ACTION POSTRUN:
(******************************************************************************)
(********** Release of PostRun - Move System to Shutdown task   ***************)
(******************************************************************************)
CallPostRunNr_no_u16 := CallPostRunNr_no_u16 + 1;

(* Release Postrun after 5 sec *)
IF (CallPostRunNr_no_u16 > 500) THEN
    bds_sys_releasePostRunProlong(); (* transitions system state from POSTRUN to SHUTDOWN *)
END_IF
END_ACTION

ACTION READ_PARAMETERS:
(******************************************************************************)
(************************ Debug Manager  **************************************)
(******************************************************************************)
PRG_DebugManager();
(******************************************************************************)
(************************ NVM Config.  ****************************************)
(******************************************************************************)
PRG_NVMConfig();
END_ACTION

ACTION RUN:
(******************************************************************************)
(**************************** CAN Wakeup Handling   ***************************)
(******************************************************************************)
(* resetInfo_s.rbr_UserDefined_u32 = 0x01 means that the Wakeup has happened via CAN via CAN Channel 1 *)
(* resetInfo_s.rbr_UserDefined_u32 = 0x04 means that the Wakeup has happened via CAN via CAN Channel 4 *)
IF ((16#01 = INIT_PRG.ResetInfo_struc.rbr_UserDefined_u32) OR (16#04 = INIT_PRG.ResetInfo_struc.rbr_UserDefined_u32)) THEN
    bds_sys_cancelAltWakeup(); (* forces system state to go to POSTRUN *)
END_IF
END_ACTION

ACTION STARTLOCK:
StartRelease_st_b := TRUE;
END_ACTION

END_PROGRAM

// BODAS_RC18_12_40/Application/01 MainTask/03 Communication/00 CAN/PRG_CANOut
(*********************************************************************************************************************
 *     __   __   ___  ___           __   __        __   __  ___
 *   /_ / /  / /__  /    /__/     /_ / /_   |_ / /_ / /  /  /  /__/
 *  /__/ /__/ __ / /__  /  /     /  | /__  /  | /  | /__/  /  /  /
 *
 * Project: Hello World for ml290.rts
 *
 * Program: PRG_CANOut
 *
 * Author:  
 *
 * Description:
 * Interface for CAN Transmitting
 *
 * (c) Copyright by BOSCH REXROTH AG, all rights reserved
 *
 *********************************************************************************************************************)
PROGRAM PRG_CANOut
VAR
    (* Buffer for rx databoxes *)
    CAN1RxData_astruc   : ARRAY[1..2] OF bds_can_DataboxData_ts;
    CAN2RxData_astruc   : ARRAY[1..5] OF bds_can_DataboxData_ts;
    bds_IPduGrpVctr_au8 : ARRAY[0..7] OF USINT;
    retSet_u16          : UINT;
    retStrt_u16         : UINT;
    data_au8            : ARRAY[1..8] OF USINT;
    dataTx_au8          : ARRAY[1..8] OF USINT; (* data ARRAY FOR CAN legacy data*)
    sigData_au8         : ARRAY[1..8] OF USINT; (* data ARRAY FOR CAN signal based data*)
END_VAR
VAR_INPUT
    i_statusNvmIni_u16  : UINT;
    i_iPmpFwdAct_mA_u16 : UINT;
    i_iPmpFwdSet_mA_u16 : UINT;
    i_CtrlValve_u8      : USINT;
    i_rxActEngPercTq_u8 : USINT;
    i_vWhlSpd_kph_u16   : INT;
    i_uPmpSnsr_mV_u16   : UINT;
    i_frqVehSnsr_Hz_u32 : UDINT;
    i_anValue_perc_u8   : USINT;
    i_stBrkSwt_u8       : USINT;
END_VAR
VAR_OUTPUT
END_VAR

(* ----------------------------------------------------------------------- *)
(* --- CAN legacy transmit --- *)
(* ----------------------------------------------------------------------- *)
(* Send a cyclic STD CAN message ON CAN1 when in OsMain *)
bds_can_sendData(bds_can_Chnl_te.BDS_CAN_1_D, 16#2, BDS_CAN_STD_DU8, 0, 0);
(* SnsrInp1 Tx *)
dataTx_au8[1] := UINT_TO_USINT(i_uPmpSnsr_mV_u16);
dataTx_au8[2] := UINT_TO_USINT(SHR(i_uPmpSnsr_mV_u16, 8));
dataTx_au8[3] := i_stBrkSwt_u8;
dataTx_au8[4] := UDINT_TO_USINT(i_frqVehSnsr_Hz_u32);
dataTx_au8[5] := UDINT_TO_USINT(SHR(i_frqVehSnsr_Hz_u32, 8));
dataTx_au8[6] := UDINT_TO_USINT(SHR(i_frqVehSnsr_Hz_u32, 16));
dataTx_au8[7] := UDINT_TO_USINT(SHR(i_frqVehSnsr_Hz_u32, 24));
dataTx_au8[8] := i_anValue_perc_u8; (* to test if 0x18FF1128 is received - legacy*)

IF (0 = bds_can_sendData(bds_can_Chnl_te.BDS_CAN_2_D, 16#18FF2703, BDS_CAN_EXD_DU8, 8, ADR(dataTx_au8))) THEN
    (* ok, message is buffered and will be sent as fast as possible *)
    ;
END_IF

(* ELSE: error *)
(* Outp1 Tx message from CAN dbc *)
(* Output currents *)
dataTx_au8[1] := UINT_TO_USINT(i_iPmpFwdAct_mA_u16);         (* LSB *)
dataTx_au8[2] := UINT_TO_USINT(SHR(i_iPmpFwdAct_mA_u16, 8)); (* MSB *)
dataTx_au8[3] := UINT_TO_USINT(i_iPmpFwdSet_mA_u16);
dataTx_au8[4] := UINT_TO_USINT(SHR(i_iPmpFwdSet_mA_u16, 8));
dataTx_au8[5] := i_CtrlValve_u8;
dataTx_au8[6] := TO_USINT(GlobalVariables.PrmAsw_gstruc.listCtrlVlv_enu);                   (* to test if the list DID C002 is received *)
dataTx_au8[7] := TO_USINT(INT_TO_WORD(GlobalVariables.PrmAsw_gstruc.nrCogs_s16) AND 16#FF); (* to test if the no. of cogs DID C003 is received *)
dataTx_au8[8] :=
    i_rxActEngPercTq_u8; (* to test if ComConf_ComSignal_ComSignal_ActualEngPercentTorque_xRx is received *)

IF (0 = bds_can_sendData(bds_can_Chnl_te.BDS_CAN_2_D, 16#18FF2603, BDS_CAN_EXD_DU8, 8, ADR(dataTx_au8))) THEN
    (* ok, message is buffered and will be sent as fast as possible *)
    ;
END_IF

(* else: error *)
(* ----------------------------------------------------------------------- *)
(* --- CAN signal based transmit --- *)
(* ----------------------------------------------------------------------- *)
(* CCVS message FROM CAN dbc - out OF the 100 ms loop *)
(* Vehicle Speed *)
sigData_au8[1] := UINT_TO_USINT(i_vWhlSpd_kph_u16);
sigData_au8[2] := UINT_TO_USINT(SHR(i_vWhlSpd_kph_u16, 8));

IF (0 = bds_can_sendSignal(ComConf_ComSignal_ComSignal_WheelBasedVehicleSpeed_xTx, ADR(sigData_au8), 0)) THEN
    (* ok,message is sent on bus with updated signal data *)
    ;
END_IF

(* Parking Brake (Control Valve) *)
sigData_au8[1] := i_CtrlValve_u8;

IF (0 = bds_can_sendSignal(ComConf_ComSignal_ComSignal_ParkingBrakeSwitch_xTx, ADR(sigData_au8), 0)) THEN
    (* ok,message is sent on bus with updated signal data *)
    ;
END_IF

END_PROGRAM

// BODAS_RC18_12_40/Application/01 MainTask/11 Parameters/Programs/PRG_NVMConfig
(*********************************************************************************************************************
 *     __   __   ___  ___           __   __        __   __  ___
 *   /_ / /  / /__  /    /__/     /_ / /_   |_ / /_ / /  /  /  /__/
 *  /__/ /__/ __ / /__  /  /     /  | /__  /  | /  | /__/  /  /  /
 *
 * Project: Hello World for ml290.rts
 *
 * Program: PRG_NVMConfig
 *
 * Author:  
 *
 * Description:
 * Interface for Paramters
 *
 * (c) Copyright by BOSCH REXROTH AG, all rights reserved
 *
 *********************************************************************************************************************)
PROGRAM PRG_NVMConfig
VAR
    status_u16 : UINT;
END_VAR

;

END_PROGRAM

// BODAS_RC18_12_40/Application/01 MainTask/02 Outputs/PRG_Outputs
(*********************************************************************************************************************
*    __   __   ___  ___           __   __        __   __  ___
*   /_ / /  / /__  /    /__/     /_ / /_   |_ / /_ / /  /  /  /__/
*  /__/ /__/ __ / /__  /  /     /  | /__  /  | /  | /__/  /  /  /
*
* Project: Hello World for ml290.rts
*
* Program: PRG_Outputs
*
* Author: 
*
* Description:
* Interface for the hardware outputs to the application
*
* (c) Copyright by BOSCH REXROTH AG, all rights reserved
*
*********************************************************************************************************************)
PROGRAM PRG_Outputs
VAR_INPUT
    i_UPumpSensr_mV_u16 : UINT;
END_VAR
VAR
    diagParam_s             : bds_outCmn_diagParam_ts;
    bds_outPwm_retGet_s     : bds_outPwm_get_ts; (* PWM output status *)
    no_UBatt_mV_u16         : UINT;
    st_FlgInhActive_b       : BOOL;
    st_FlgUBatLowDetd_b     : BOOL;
    st_FlgUBatLowDetdPrev_b : BOOL;
    st_FlgOutpLocked_b      : BOOL;
    st_FlgUnderUbat_b       : BOOL;
    st_FlgRstInh_b          : BOOL;
    st_FlgRstLowBatt_b      : BOOL;
    no_NrCycDebRst_u16      : UINT;
    no_CurrentK07_mA_u16    : UINT;
    iPmpFwdSet_mA_u16       : UINT;
    st_CurStK07_u8          : USINT;
    no_UPumpSensr_mV_u16    : UINT;
    st_CtrlValve_u8         : USINT;
    st_BrkSwt_u8            : USINT;
    MngInh_struc            : struc_MngInhb;
    PHMDL_CHNL1             : UINT := (UDINT_TO_UINT(PHMDL) OR UDINT_TO_UINT(CHNL1));
END_VAR
VAR CONSTANT
    st_ENotOk_cby    : BYTE := 16#01;
    st_StdHigh_cby   : BYTE := 16#01;
    st_StdLow_cby    : BYTE := 16#00;
    st_StdActive_cby : BYTE := 16#01;
    st_StdIdle_cby   : BYTE := 16#00;
    st_StdOn_cby     : BYTE := 16#00;
    st_StdOff_cby    : BYTE := 16#01;
END_VAR

(* Inhibit handling *)
ACT_HandleInhibit();
(* PropValve - read actual current *)
bds_outPwm_retGet_s := bds_outPwm_get(bds_outPwm_signal_te.bds_outPwm_K07_E);

(* check return state of BDS-Function call *)
IF (bds_outCmn_ok_E = bds_outPwm_retGet_s.statusApi_e) THEN
    (* Call successful, signal is valid *)
    ;
ELSE
    (* error handling *)
    no_CurrentK07_mA_u16 := bds_outPwm_retGet_s.iAct_mA_u16;
END_IF

(* Calculate set current *)
(* PropValve [K07]= PmpSensor [K52] * Factor [parameter DID 0xC001] *)
iPmpFwdSet_mA_u16 := i_UPumpSensr_mV_u16 * INT_TO_UINT(GlobalVariables.PrmAsw_gstruc.fctPmp_s16);

(* Calculate set state *)
(* CtrlValve [K12] = BrkSwitch [K78] | List [DID 0xC002] *)
CASE (GlobalVariables.PrmAsw_gstruc.listCtrlVlv_enu) OF
enu_listCtrlVlv.st_fctOff_cenu: st_CtrlValve_u8   := st_StdIdle_cby;
enu_listCtrlVlv.st_fctOnPos_cenu: st_CtrlValve_u8 := st_BrkSwt_u8;
enu_listCtrlVlv.st_fctOnNeg_cenu: IF (NOT (0 = st_BrkSwt_u8)) THEN
        st_CtrlValve_u8 := st_StdIdle_cby;
    ELSE
        st_CtrlValve_u8 := st_StdActive_cby;
    END_IF
    ELSE
        ;
END_CASE

(* ----------------------------------------------------------------------- *)
(* --- Set outputs ---*)
(* ----------------------------------------------------------------------- *)
(* Set outputs only when inhibit is not active *)
(* PropValve *)
bds_outPwm_cfgMode(bds_outPwm_signal_te.bds_outPwm_K07_E, bds_outMode_CLCC_E);   (* Configure K07 as closed loop current control *)
bds_outPwm_setCurrent(bds_outPwm_signal_te.bds_outPwm_K07_E, iPmpFwdSet_mA_u16); (* Set current set point for proportional valve *)
(* CtrlValve *)
bds_outDig_set(bds_outDig_signal_te.bds_outDig_K13_E, (st_CtrlValve_u8 > 0));
(* Safout *)
bds_out_po_cfg(bds_out_po_signal_te.K09, STD_ON);                                                (* Configure K09 as closed loop current control *)
bds_out_po_cfg(bds_out_po_signal_te.K73, STD_ON);                                                (* Configure K73 as closed loop current control *)
bds_safout(PHMDL_CHNL1, bds_out_po_signal_te.K09, GlobalVariables.PrmAsw_gstruc.iSpSafout1_u16); (* Safout - HS1 *)
bds_safout(PHMDL_CHNL1, bds_out_po_signal_te.K73, GlobalVariables.PrmAsw_gstruc.iSpSafout2_u16); (* Safout - HS2 *)

ACTION ACT_HandleInhibit:
(* Monitor battery voltage AND state OF inhibit            *
 * reset inhibit in CASE it was activated BY under voltage *
*)
(* Invert logic of flgStInhb_u8 *)
st_FlgInhActive_b := NOT( PRG_Inputs.st_FlgStInhb_u8 > 0 );

bds_sys_aiv(bds_sys_aiv_signal_te.UBAT_MON, ADR(no_UBatt_mV_u16));  (* battery supply voltage *)   

IF( no_UBatt_mV_u16 < 7000 ) THEN (* under voltage detection if the battery voltage is less than 7V *)
  st_FlgUnderUbat_b := TRUE;
END_IF
      
st_FlgUBatLowDetd_b := ( ( st_FlgInhActive_b )OR (6500  >  no_UBatt_mV_u16 ) );

(* Inhibit Reset (i.e. release outputs again after emergency stop) *)
st_FlgRstInh_b :=	st_FlgInhActive_b                   AND  (* Inhibit is active -> Outputs are disabled *)
					( 9000 <  no_UBatt_mV_u16 )         AND  (* Voltage is greater than x V *)
					( 0    =  PRG_Inputs.st_K21Inh_u8 ) AND  (* Inhibit inputs are in a legitimate state *)
					( 0    <> PRG_Inputs.st_K22Inh_u8 );     (* Inhibit inputs are in a legitimate state *)
					
(* Low Battery Reset (i.e. release outputs after low battery was detected) *)
st_FlgRstLowBatt_b :=	st_FlgInhActive_b           AND  (* Inhibit is not active *)  
						st_FlgOutpLocked_b          AND  (* Outputs are locked *)
						( 9000 < no_UBatt_mV_u16 );      (* Voltage is greater than x V *)
						
						
(* Debounce Reset *)
IF( st_FlgRstInh_b OR st_FlgRstLowBatt_b ) THEN  
	no_NrCycDebRst_u16 := no_NrCycDebRst_u16 + 1;
END_IF					


IF( 5 < no_NrCycDebRst_u16 ) THEN
	(* Reset inhibit (enables the output again) *)	
	bds_sys_resetINH();
	
	(* Re-Configure K08 as power supply FOR K13 Control valve *)
	diagParam_s.diFullDiag_l     := TRUE;
	diagParam_s.diCntlAndDiag_l  := FALSE;
	diagParam_s.diOpenLoadDetn_l := TRUE;
	diagParam_s.diNonHotSCDetn_l := FALSE;
	
	bds_outPwm_cfgDiag(bds_outPwm_signal_te.bds_outPwm_K08_E, diagParam_s);
	bds_outPwm_setDutyCycle(bds_outPwm_signal_te.bds_outPwm_K08_E, 1000);
	
	st_FlgUnderUbat_b  := FALSE;
	no_NrCycDebRst_u16 := 0;

ELSE
	;	
END_IF
END_ACTION

ACTION ACT_InitOutputs:
diagParam_s.diCntlAndDiag_l := TRUE; (* disable outputs *)
(* Disable unused proportional outputs *)
(*bds_outPwm_cfgDiag(bds_outPwm_signal_te.bds_outPwm_K07_E, diagParam_s);*) (* used FOR PropValve *)
(*bds_outPwm_cfgDiag(bds_outPwm_signal_te.bds_outPwm_K09_E, diagParam_s);*) (* Safout HS1 *)
(*bds_outPwm_cfgDiag(bds_outPwm_signal_te.bds_outPwm_K73_E, diagParam_s);*) (* Safout HS2 *)
(*bds_outPwm_cfgDiag(bds_outPwm_signal_te.bds_outPwm_K08_E, diagParam_s);*) (* used as power supply for Control valve *)
bds_outPwm_cfgDiag(bds_outPwm_signal_te.bds_outPwm_K29_E, diagParam_s);
bds_outPwm_cfgDiag(bds_outPwm_signal_te.bds_outPwm_K17_E, diagParam_s);
bds_outPwm_cfgDiag(bds_outPwm_signal_te.bds_outPwm_A32_E, diagParam_s);
bds_outPwm_cfgDiag(bds_outPwm_signal_te.bds_outPwm_A47_E, diagParam_s);
bds_outPwm_cfgDiag(bds_outPwm_signal_te.bds_outPwm_A31_E, diagParam_s);
bds_outPwm_cfgDiag(bds_outPwm_signal_te.bds_outPwm_A48_E, diagParam_s);
bds_outPwm_cfgDiag(bds_outPwm_signal_te.bds_outPwm_A46_E, diagParam_s);
bds_outPwm_cfgDiag(bds_outPwm_signal_te.bds_outPwm_A33_E, diagParam_s);
bds_outPwm_cfgDiag(bds_outPwm_signal_te.bds_outPwm_A34_E, diagParam_s);
bds_outPwm_cfgDiag(bds_outPwm_signal_te.bds_outPwm_A51_E, diagParam_s);
bds_outPwm_cfgDiag(bds_outPwm_signal_te.bds_outPwm_A35_E, diagParam_s);
bds_outPwm_cfgDiag(bds_outPwm_signal_te.bds_outPwm_A53_E, diagParam_s);
bds_outPwm_cfgDiag(bds_outPwm_signal_te.bds_outPwm_A52_E, diagParam_s);
bds_outPwm_cfgDiag(bds_outPwm_signal_te.bds_outPwm_A54_E, diagParam_s);
bds_outPwm_cfgDiag(bds_outPwm_signal_te.bds_outPwm_K16_E, diagParam_s);
(*bds_outPwm_cfgDiag(bds_outPwm_signal_te.bds_outPwm_K14_E, diagParam_s);*) (* Safout LS *)
bds_outPwm_cfgDiag(bds_outPwm_signal_te.bds_outPwm_K15_E, diagParam_s);
bds_outPwm_cfgDiag(bds_outPwm_signal_te.bds_outPwm_A19_E, diagParam_s);
bds_outPwm_cfgDiag(bds_outPwm_signal_te.bds_outPwm_A05_E, diagParam_s);
bds_outPwm_cfgDiag(bds_outPwm_signal_te.bds_outPwm_A20_E, diagParam_s);
bds_outPwm_cfgDiag(bds_outPwm_signal_te.bds_outPwm_A09_E, diagParam_s);
bds_outPwm_cfgDiag(bds_outPwm_signal_te.bds_outPwm_A02_E, diagParam_s);
bds_outPwm_cfgDiag(bds_outPwm_signal_te.bds_outPwm_A17_E, diagParam_s);
bds_outPwm_cfgDiag(bds_outPwm_signal_te.bds_outPwm_K51_E, diagParam_s);
bds_outPwm_cfgDiag(bds_outPwm_signal_te.bds_outPwm_K12_E, diagParam_s);
bds_outPwm_cfgDiag(bds_outPwm_signal_te.bds_outPwm_A03_E, diagParam_s);
bds_outPwm_cfgDiag(bds_outPwm_signal_te.bds_outPwm_A18_E, diagParam_s);
bds_outPwm_cfgDiag(bds_outPwm_signal_te.bds_outPwm_A08_E, diagParam_s);
bds_outPwm_cfgDiag(bds_outPwm_signal_te.bds_outPwm_A07_E, diagParam_s);
bds_outPwm_cfgDiag(bds_outPwm_signal_te.bds_outPwm_K80_E, diagParam_s);
bds_outPwm_cfgDiag(bds_outPwm_signal_te.bds_outPwm_K81_E, diagParam_s);
bds_outPwm_cfgDiag(bds_outPwm_signal_te.bds_outPwm_K82_E, diagParam_s);
bds_outPwm_cfgDiag(bds_outPwm_signal_te.bds_outPwm_K83_E, diagParam_s);
(* Disable unused digital outputs *)
(*bds_outDig_cfgDiag(bds_outDig_K13_E, diagParam_s);*) (* used for CtrlValve *)
bds_outDig_cfgDiag(bds_outDig_signal_te.bds_outDig_A04_E, diagParam_s);
bds_outDig_cfgDiag(bds_outDig_signal_te.bds_outDig_A10_E, diagParam_s);
bds_outDig_cfgDiag(bds_outDig_signal_te.bds_outDig_A50_E, diagParam_s);
bds_outDig_cfgDiag(bds_outDig_signal_te.bds_outDig_A56_E, diagParam_s);
bds_outDig_cfgDiag(bds_outDig_signal_te.bds_outDig_A11_E, diagParam_s);
bds_outDig_cfgDiag(bds_outDig_signal_te.bds_outDig_A55_E, diagParam_s);
bds_outDig_cfgDiag(bds_outDig_signal_te.bds_outDig_A01_E, diagParam_s);
bds_outDig_cfgDiag(bds_outDig_signal_te.bds_outDig_A06_E, diagParam_s);
bds_outDig_cfgDiag(bds_outDig_signal_te.bds_outDig_A16_E, diagParam_s);
bds_outDig_cfgDiag(bds_outDig_signal_te.bds_outDig_A58_E, diagParam_s);
bds_outDig_cfgDiag(bds_outDig_signal_te.bds_outDig_A49_E, diagParam_s);
bds_outDig_cfgDiag(bds_outDig_signal_te.bds_outDig_K84_E, diagParam_s);
bds_outDig_cfgDiag(bds_outDig_signal_te.bds_outDig_K85_E, diagParam_s);
bds_outDig_cfgDiag(bds_outDig_signal_te.bds_outDig_K86_E, diagParam_s);
bds_outDig_cfgDiag(bds_outDig_signal_te.bds_outDig_K87_E, diagParam_s); (* for the visualisation in BODAS-service App --> I/O *)
(* Configure K08 as power supply for K13 Control valve *)
diagParam_s.diFullDiag_l     := TRUE;
diagParam_s.diCntlAndDiag_l  := FALSE;
diagParam_s.diOpenLoadDetn_l := TRUE;
diagParam_s.diNonHotSCDetn_l := FALSE;
bds_outPwm_cfgDiag(bds_outPwm_signal_te.bds_outPwm_K08_E, diagParam_s);
bds_outPwm_setDutyCycle(bds_outPwm_signal_te.bds_outPwm_K08_E, 1000);
END_ACTION

END_PROGRAM

// BODAS_RC18_12_40/Application/01 MainTask/01 Inputs/PRG_Inputs
(*********************************************************************************************************************
 *     __   __   ___  ___           __   __        __   __  ___
 *   /_ / /  / /__  /    /__/     /_ / /_   |_ / /_ / /  /  /  /__/
 *  /__/ /__/ __ / /__  /  /     /  | /__  /  | /  | /__/  /  /  /
 *
 * Project: Hello World for ml290.rts
 *
 * Program: PRG_Inputs
 *
 * Author:  
 *
 * Description:
 * Interface for the hardware inputs to the application
 *
 * (c) Copyright by BOSCH REXROTH AG, all rights reserved
 *
 *********************************************************************************************************************)
PROGRAM PRG_Inputs
VAR_INPUT
    i_TaskCycleTime_ms_u16 : UINT;
END_VAR
VAR
    st_K21Inh_u8           : USINT;
    st_K22Inh_u8           : USINT;
    st_FlgStInhb_u8        : USINT;
    bds_inPwm_getFrqPwm_s  : bds_inPwm_frqMeasmt_ts;
    FrqP_Hz_10_u32         : UDINT;                (* frequency [0.1Hz] *)
    Tmp_u32                : UDINT;                (* temporary *)
    stPmpSnsrU_struc       : bds_inU_measmt_ts;    (*structure FOR Pump sensor voltage measurement *)
    uPmpSnsr_mV_u16        : UINT;                 (* voltage [mV], ECU pin K52 *)
    stPmpSnsrSigInvldErr_e : bds_dsmCmn_fltLvl_te; (* status of error: PmpSnsr *)
    (* K78 � DIG, BrkSwitch - read as AIV *)
    stBrkSwtU_struc       : bds_inU_measmt_ts;    (* structure FOR Brake switch voltage measurement *)
    uBrkSwt_mV_u16        : UINT;                 (* voltage [mV], ECU pin K78 *)
    stBrkSwt_u8           : USINT;                (* status OF break switch, ECU pin K78 *)
    stBrkSwtSigInvldErr_e : bds_dsmCmn_fltLvl_te; (* status OF error: BrkSwt *)
    (* K54_VI � FREQ, VehSensor *)
    stVehSnsrFrq_struc : bds_inPwm_frqMeasmt_ts; (*structure FOR vehicle sensor frequency measurement *)
    frqVehSnsr_Hz_u32  : UDINT;                  (* frequency [Hz], ECU pin K54_VI *)
    vWhlSpd_kph_u16    : UINT;                   (* vehicle speed [km/h] *)
    (* K37 and K41 - DST Sensor *)
    SpdSnsrDST1_struc         : bds_snsrDst_getSpdAndDir_ts;
    SpdSnsrDST1_inst_enu      : bds_snsrDst_inst_te;
    SpdSnsrDST1_dRpm_u32      : UDINT;
    SpdSnsrDST1_rotDir_enu    : bds_snsrDst_dir_te;
    SpdSnsrDST1Temp_struc     : bds_snsrDst_getTemp_ts;
    SpdSnsrDST1_temp_degC_s32 : DINT;
    (* PR4SENTSnsr - BDL *)
    PR4Snsr_getP_struc : bds_snsrPr4_getPressure_ts;
    PR4SnsrP_u16       : UINT;
    PR4Snsr_getT_struc : bds_snsrPr4_getTemp_ts;
    PR4SnsrT_s32       : DINT;
END_VAR
VAR_OUTPUT
    o_T15_st_u8 : USINT;
END_VAR
VAR CONSTANT
    PI_no_100_u16         : UINT := 314;
    Rad_m_u16             : UINT := 1;
    PR4SnsrPCalcY1Fact    : UINT := 193;
    PR4SnsrPCalcY2Y1Fact  : UINT := 3703;
    PR4SnsrPCalcX2X1Range : UINT := 50;
    PR4SnsrTCalcX1Fact    : UINT := 200;
    PR4SnsrTCalcY2Y1Fact  : UINT := 4088;
    PR4SnsrTCalcX2X1Range : UINT := 511;
END_VAR

(* Inhibit active at low battery voltage *)
(* get the states of inhibits*)
bds_in_di(bds_in_di_signal_te.K21, ADR(st_K21Inh_u8));
bds_in_di(bds_in_di_signal_te.K22, ADR(st_K22Inh_u8));
(* get a state of the inhibit signal *)
bds_sys_di(bds_sys_di_signal_te.ST_INH, ADR(st_FlgStInhb_u8));
(* get state of T15 *)
bds_sys_getT15(ADR(o_T15_st_u8));
(* ----------------------------------------------------------------------- *)
(* --- Read inputs ---*)
(* ----------------------------------------------------------------------- *)
(* PumpSensor - voltage *)
(* Get the voltage value of input signal K52 *)
stPmpSnsrU_struc := bds_inU_get(bds_inU_signal_te.bds_inU_K52_E);

(* get the measured voltage on selected input signal *)
IF (bds_inCmn_ok_E = stPmpSnsrU_struc.status_e) THEN
    (* save the actual voltage into local variable *)
    uPmpSnsr_mV_u16 := stPmpSnsrU_struc.u_mV_u16;
    (* Report no error *)
    stPmpSnsrSigInvldErr_e := bds_dsmCmn_fltLvl_0_Perc_e;
ELSE
    (* Report an error *)
    stPmpSnsrSigInvldErr_e := bds_dsmCmn_fltLvl_100_Perc_e;
    (* BrkSwitch - as digital *)
    (* Get the voltage value of input signal K78 *)
    stBrkSwtU_struc := bds_inU_get(bds_inU_signal_te.bds_inU_K78_E);

    (* get the measured voltage on selected input signal *)
    IF (bds_inCmn_ok_E = stBrkSwtU_struc.status_e) THEN
        (* save the actual voltage into local variable *)
        uBrkSwt_mV_u16 := stBrkSwtU_struc.u_mV_u16;
        (* Report no error *)
        stBrkSwtSigInvldErr_e := bds_dsmCmn_fltLvl_0_Perc_e;
    ELSE
        (* Report an error *)
        stBrkSwtSigInvldErr_e := bds_dsmCmn_fltLvl_100_Perc_e;
    END_IF
END_IF

(* VehSensor - frequency *)
(* Get the pwm frequency value of input signal K54 *)
stVehSnsrFrq_struc := bds_inPwm_getFrq(bds_inPwm_signal_te.bds_inPwm_K54_E);

(* get the actual pwm frequency on selected input signal *)
IF (bds_inCmn_ok_E = stVehSnsrFrq_struc.status_e) THEN
    (* save the actual pwm times AND counter into local variable *)
    FrqP_Hz_10_u32 := stVehSnsrFrq_struc.frq_dHz_u32;
    (*convert into Hz *)
    FrqP_Hz_10_u32 := FrqP_Hz_10_u32 + 5;  (* rounding the value *)
    Tmp_u32        := FrqP_Hz_10_u32 / 10; (* convert in Hz *)
    FrqP_Hz_10_u32 := MIN(Tmp_u32, 16#FFFF);
ELSE
    (* Report no error *)
    (* stVehSnsrSigInvldErr_u16 := BDS_DSM_FAULT_PERCENT_00_DU8; *)
END_IF

(* ----------------------------------------------------------------------- *)
(* --- BODASDriver library (BDL) *)
(* ----------------------------------------------------------------------- *)
(* ----------------------------------------------------------------------- *)
(* --- Rotation Speed Sensor (DST)*)
(* ----------------------------------------------------------------------- *)
SpdSnsrDST1_struc := bds_snsrDst_getSpdAndDir(bds_snsrDst_inst_te.SpdSnsr_E);

(* check the return status of API function call *)
IF (bds_snsrDst_ok_E = SpdSnsrDST1_struc.statusApi_e) THEN
    (* save the actual wheel speed and rotation direction *)
    SpdSnsrDST1_dRpm_u32   := SpdSnsrDST1_struc.spd_dRpm_u32;
    SpdSnsrDST1_rotDir_enu := SpdSnsrDST1_struc.dir_e;
END_IF

(* BDL API function call for temperature *)
SpdSnsrDST1Temp_struc := bds_snsrDst_getTemp(bds_snsrDst_inst_te.SpdSnsr_E);

(* check the return status of API function call *)
IF (bds_snsrDst_ok_E = SpdSnsrDST1Temp_struc.statusApi_e) THEN
    (* save the actual temperature in degree celsius *)
    SpdSnsrDST1_temp_degC_s32 := SpdSnsrDST1Temp_struc.temp_degC_s32;
END_IF

(***************************************************************)
(*  PR4SENTSnsr                              				   *)
(***************************************************************)
(* BDL API function call to get pressure *)
PR4Snsr_getP_struc := bds_snsrPr4_getPressure(bds_snsrPr4_inst_te.pSnsr_E);

(* check the return status of API function call *)
IF (bds_snsrPr4_ok_E = PR4Snsr_getP_struc.stsApi_e) THEN
    (* save the actual wheel speed and rotation direction *)
    PR4SnsrP_u16 := PR4Snsr_getP_struc.pressure_dBar_u16;
END_IF

(* BDL API function call to get temperature*)
PR4Snsr_getT_struc := bds_snsrPr4_getTemp(bds_snsrPr4_inst_te.pSnsr_E);

(* check the return status of API function call *)
IF (bds_snsrPr4_ok_E = PR4Snsr_getT_struc.stsApi_e) THEN
    (* save the actual temperature in degree celsius *)
    PR4SnsrT_s32 := PR4Snsr_getT_struc.temp_degC_s32;
END_IF

(* ----------------------------------------------------------------------- *)
(* --- Processing of inputs and outputs ---*)
(* ----------------------------------------------------------------------- *)
(* Brake switch status evaluation: Maximum threshold 2.2V and Minimum Threshold 0.8V *)
IF ((uBrkSwt_mV_u16 > 2200) AND (uBrkSwt_mV_u16 < 5200)) THEN
    stBrkSwt_u8 := 1;
ELSIF (uBrkSwt_mV_u16 < 800) THEN
    stBrkSwt_u8 := 0;
ELSE
    (* do nothing *)
    ;
END_IF

(* Calculate vehicle speed *)
Tmp_u32 := frqVehSnsr_Hz_u32 * 3600 * 2 * PI_no_100_u16 * Rad_m_u16 / 1000 / 100;
(*Tmp_r := ROUND((float)frqVehSnsr_Hz_u32 * (float32)3600 * ((float32)2 * Pi_DF32 * (float32)r_DU16) / (float32)1000);
*)
(* Vehicle speed [CCVS] based on frq. [K54_VI] depending on #cogs [0xC003] *)
vWhlSpd_kph_u16 := DINT_TO_UINT(UDINT_TO_DINT(Tmp_u32) / GlobalVariables.PrmAsw_gstruc.nrCogs_s16);

ACTION ACT_InitInputs:
(* activate FI *)
//bds_in_fi_cfg(bds_in_fi_signal_te.K54_VI, STD_OFF);
(* DST Sensor *)
(* BDL API FUNCTION call TO configure DST sensor instance *)
bds_snsrDst_cfgSpdAndDir(bds_snsrDst_inst_te.SpdSnsr_E, 75);
END_ACTION

END_PROGRAM

// BODAS_RC18_12_40/Application/01 MainTask/03 Communication/00 CAN/PRG_CANIn
(*********************************************************************************************************************
 *     __   __   ___  ___           __   __        __   __  ___
 *   /_ / /  / /__  /    /__/     /_ / /_   |_ / /_ / /  /  /  /__/
 *  /__/ /__/ __ / /__  /  /     /  | /__  /  | /  | /__/  /  /  /
 *
 * Project: Hello World for ml290.rts
 *
 * Program: PRG_CANIn
 *
 * Author:  
 *
 * Description:
 * Interface for CAN Receiving
 *
 * (c) Copyright by BOSCH REXROTH AG, all rights reserved
 *
 *********************************************************************************************************************)
PROGRAM PRG_CANIn
VAR
	(* Buffer for rx databoxes *)
	CAN1RxData_astruc : ARRAY[1..2] OF bds_can_DataboxData_ts;
	CAN2RxData_astruc : ARRAY[1..5] OF bds_can_DataboxData_ts;
	
	sigData_au8 : ARRAY[1..8] OF USINT;			        (* data ARRAY FOR CAN signal based data*)
END_VAR

VAR_OUTPUT
	o_rxActEngPercTq_u8 : USINT;
END_VAR

(* ----------------------------------------------------------------------- *)
(* --- CAN signal based receive --- *)
(* ----------------------------------------------------------------------- *)

IF( 0 = bds_can_receiveSignal( ComConf_ComSignal_ComSignal_ActualEngPercentTorque_xRx, ADR(sigData_au8), 0 ) ) THEN

	  (* Data is stored in sigData_au8. *)
	  (* The signal ActualEngPercentTorque is 1 byte so copy the 1st byte and update the test variable.*)
	  o_rxActEngPercTq_u8 := sigData_au8[1];
END_IF

END_PROGRAM

// BODAS_RC18_12_40/Application/01 MainTask/20_Errors/PRG_HandleErrors
(*********************************************************************************************************************
 *     __   __   ___  ___           __   __        __   __  ___
 *   /_ / /  / /__  /    /__/     /_ / /_   |_ / /_ / /  /  /  /__/
 *  /__/ /__/ __ / /__  /  /     /  | /__  /  | /  | /__/  /  /  /
 *
 * Project: Hello World for ml290.rts
 *
 * Program: PRG_HandleErrors
 *
 * Author:  
 *
 * Description:
 * Error Handling
 *
 * (c) Copyright by BOSCH REXROTH AG, all rights reserved
 *
 *********************************************************************************************************************)
PROGRAM PRG_HandleErrors
VAR_INPUT
    i_stPmpSnsrSigInvldErr_e : bds_dsmCmn_fltLvl_te;
    i_stBrkSwtSigInvldErr_e  : bds_dsmCmn_fltLvl_te;
    i_uPmpSnsr_mV_u16        : UINT;
    i_frqVehSnsr_Hz_u32      : UINT;
    i_iPmpFwdAct_mA_u16      : UINT;
    i_vWhlSpd_kmh_u16        : UINT;
END_VAR
VAR
    chkResult_e : bds_dsmCmn_fltLvl_te;
    (* DFC type definitions *)
    DFC_bds_TiUpDwn0x8A03_ts : DFC_bds_TiUpDwn0x8A03;
    DFC_bds_TiUpDwn0x8A02_ts : DFC_bds_TiUpDwn0x8A02;
    DFC_bds_TiInRow0x8B02_ts : DFC_bds_TiInRow0x8B02;
    DFC_bds_TiUpDwn0x8A01_ts : DFC_bds_TiUpDwn0x8A01;
    DFC_bds_TiInRow0x8B01_ts : DFC_bds_TiInRow0x8B01;
    DFC_bds_TiInRow0x8B03_ts : DFC_bds_TiInRow0x8B03;
    DFC_bds_NoDeb0x8C01_ts   : DFC_bds_NoDeb0x8C01;
    DFC_bds_NoDeb0x8C03_ts   : DFC_bds_NoDeb0x8C03;
END_VAR
VAR CONSTANT
    COUNTR_DSMDEB_DU16 : UINT := 10;
END_VAR

(* ----------------------------------------------------------------------- *)
(* --- Failures - DFCs ---*)
(* ----------------------------------------------------------------------- *)
(* --- DTC 0x8A02 ---*)
(* Report error (DFC): Pump sensor signal invalidity error *)
bds_dsmDTC_updateErr(DFC_bds_TiUpDwn0x8A02_ts.DTC, i_stPmpSnsrSigInvldErr_e, (COUNTR_DSMDEB_DU16 * 1000)); (* 10msec := 10*1000usec *)
(* --- DTC 0x8B02 ---*)
(* Report error (DFC): Break switch signal invalidity error *)
bds_dsmDTC_updateErr(DFC_bds_TiInRow0x8B02_ts.DTC, i_stBrkSwtSigInvldErr_e, (COUNTR_DSMDEB_DU16 * 1000)); (* 10msec := 10*1000usec *)

(* --- DTC 0x8A01 ---*)
(* check IF error condition is fulfilled *)
IF (500 > i_uPmpSnsr_mV_u16) THEN
    (* error *)
    chkResult_e := bds_dsmCmn_fltLvl_100_Perc_e;
ELSE
    (* ok *)
    chkResult_e := bds_dsmCmn_fltLvl_0_Perc_e;
END_IF

(* report error (DFC) *)
bds_dsmDTC_updateErr(DFC_bds_TiUpDwn0x8A01_ts.DTC, chkResult_e, (COUNTR_DSMDEB_DU16 * 1000)); (*10msec := 10*1000usec*)

(* --- DTC 0x8A03 ---*)
(* check IF error condition is fulfilled *)
IF (8000 < i_frqVehSnsr_Hz_u32) THEN
    (* error *)
    chkResult_e := bds_dsmCmn_fltLvl_100_Perc_e;
ELSE
    (* ok *)
    chkResult_e := bds_dsmCmn_fltLvl_0_Perc_e;
END_IF

(* report error (DFC) *)
bds_dsmDTC_updateErr(DFC_bds_TiUpDwn0x8A03_ts.DTC, chkResult_e, (COUNTR_DSMDEB_DU16 * 1000)); (* 10msec := 10*1000usec *)

(* --- DTC 0x8B01 ---*)
(* check IF error condition is fulfilled *)
IF (3000 < i_iPmpFwdAct_mA_u16) THEN
    (* error *)
    chkResult_e := bds_dsmCmn_fltLvl_100_Perc_e;
ELSE
    (* ok *)
    chkResult_e := bds_dsmCmn_fltLvl_0_Perc_e;
END_IF

(* report error (DFC) *)
bds_dsmDTC_updateErr(DFC_bds_TiInRow0x8B01_ts.DTC, chkResult_e, (COUNTR_DSMDEB_DU16 * 1000)); (* 10msec := 10*1000usec *)

(* --- DTC 0x8B03 ---*)
IF (40 < i_vWhlSpd_kmh_u16) THEN
    (* error *)
    chkResult_e := bds_dsmCmn_fltLvl_100_Perc_e;
ELSE
    (* ok *)
    chkResult_e := bds_dsmCmn_fltLvl_0_Perc_e;
END_IF

(* report error (DFC) *)
bds_dsmDTC_updateErr(DFC_bds_TiInRow0x8B03_ts.DTC, chkResult_e, (COUNTR_DSMDEB_DU16 * 1000)); (* 10msec := 10*1000usec *)

(* --- DTC 0x8C01 ---*)
(* check IF error condition is fulfilled *)
IF (8 < GlobalVariables.PrmAsw_gstruc.fctPmp_s16) THEN
    (* error *)
    chkResult_e := bds_dsmCmn_fltLvl_100_Perc_e;
ELSE
    (* ok *)
    chkResult_e := bds_dsmCmn_fltLvl_0_Perc_e;
END_IF

(* report error (DFC) *)
bds_dsmDTC_updateErr(DFC_bds_NoDeb0x8C01_ts.DTC, chkResult_e, (COUNTR_DSMDEB_DU16 * 1000));

(* --- DTC 0x8C03 ---*)
(* check IF error condition is fullfilled *)
IF (40 < GlobalVariables.PrmAsw_gstruc.nrCogs_s16) THEN
    (* error *)
    chkResult_e := bds_dsmCmn_fltLvl_100_Perc_e;
ELSE
    (* ok *)
    chkResult_e := bds_dsmCmn_fltLvl_0_Perc_e;
END_IF

(* report error (DFC) *)
bds_dsmDTC_updateErr(DFC_bds_NoDeb0x8C03_ts.DTC, chkResult_e, (COUNTR_DSMDEB_DU16 * 1000));

ACTION ACT_InitHandleErrors:
chkResult_e := bds_dsmCmn_fltLvl_0_Perc_e;
END_ACTION

END_PROGRAM

// BODAS_RC18_12_40/Application/01 MainTask/20_Errors/PRG_ErrMemMgr
(*********************************************************************************************************************
 *     __   __   ___  ___           __   __        __   __  ___
 *   /_ / /  / /__  /    /__/     /_ / /_   |_ / /_ / /  /  /  /__/
 *  /__/ /__/ __ / /__  /  /     /  | /__  /  | /  | /__/  /  /  /
 *
 * Project: Hello World for ml290.rts
 *
 * Program: PRG_ErrMemMgr
 *
 * Author:  
 *
 * Description:
 * Handling of error memory for the workaround
 *
 * (c) Copyright by BOSCH REXROTH AG, all rights reserved
 *
 *********************************************************************************************************************)
PROGRAM PRG_ErrMemMgr
VAR
    ErrMemMgr_s           : struc_ErrMemMgr_prv;
    DFES_numEntryAvl      : UINT;
    errList_s             : bds_dsmDTC_getErrList_ts;
    dsmDTC_getStatus_s    : bds_dsmDTC_getStatus_ts;
    dfc_as                : ARRAY[0..32] OF bds_dsm_dfc_ts;
    status_u16            : UINT;
    cntrDfes_u8           : USINT;
    cntrApplBuf_u8        : USINT;
    idxActEntry_u8        : USINT;
    idxFirstEmptyEntry_u8 : USINT;
END_VAR

(* Init start value *)
ErrMemMgr_s.nrDfesEntr_u8 := 0;
(* Synchronize application buffer with DFES entries *)
ACT_GetDFESEntry();
(* Clear entries in DFES and application when maximum number of errors are exceeded i.e. 27. This shall make space for 5 new entries in DFES *)
ACT_ClrDFESEntry();

ACTION ACT_ClrDFESEntry:
(* Action: ErrMemMgr_clrDfesEntr *)
idxActEntry_u8 := ErrMemMgr_stNoEntryAvl_DU8; (* Actual index entry *)
(* delete DTCs when maximum number of entries are exceeded *)
IF ErrMemMgr_s.nrDfesEntr_u8 > ErrMemMgr_nrMaxErrEntry_DU8 THEN
    ErrMemMgr_s.tiOldStamp_u32 := 16#FFFFFFFF;
    (* delete DTCs when maximum number of entries are exceeded *)
    FOR cntrApplBuf_u8 := 0 TO ErrMemMgr_nrDfesEntries_DU8 - 1 DO
        IF (ErrMemMgr_s.tiOldStamp_u32 > ErrMemMgr_s.ErrMemMgr_savePrm_s.ErrMemMgr_prevActvDfes_as[cntrApplBuf_u8].tiStamp_min_u32) AND
           (0 < ErrMemMgr_s.ErrMemMgr_savePrm_s.ErrMemMgr_prevActvDfes_as[cntrApplBuf_u8].tiStamp_min_u32) THEN
            ErrMemMgr_s.tiOldStamp_u32 := ErrMemMgr_s.ErrMemMgr_savePrm_s.ErrMemMgr_prevActvDfes_as[cntrApplBuf_u8].tiStamp_min_u32;
            idxActEntry_u8             := cntrApplBuf_u8;
        END_IF;
    END_FOR;

    IF idxActEntry_u8 <> ErrMemMgr_stNoEntryAvl_DU8 THEN
        (* Remove oldest previously active or deactive DTC from DFES *)
        ErrMemMgr_s.status_au16[idxActEntry_u8] :=
            ErrMemMgr_s.status_au16[idxActEntry_u8] OR
            UINT_TO_WORD(bds_dsm_delError_DTC(UDINT_TO_UINT(ErrMemMgr_s.ErrMemMgr_savePrm_s
                                                                .ErrMemMgr_prevActvDfes_as[idxActEntry_u8].idxPrevActvDfes_u32)));

        ErrMemMgr_s.clrCntr_au8[idxActEntry_u8] := ErrMemMgr_s.clrCntr_au8[idxActEntry_u8] + 1;
        (* remove oldest DFC from the application buffer *)
        ErrMemMgr_s.ErrMemMgr_savePrm_s.ErrMemMgr_prevActvDfes_as[idxActEntry_u8].idxPrevActvDfes_u32 := 0;
        ErrMemMgr_s.ErrMemMgr_savePrm_s.ErrMemMgr_prevActvDfes_as[idxActEntry_u8].tiStamp_min_u32     := 0;
    END_IF;
END_IF;
END_ACTION

ACTION ACT_GetDFESEntry:
(* Action: ErrMemMgr_getDfesEntr *)
(* global variable DFES_numEntryAvl not available *)
//bds_dsm_getNumErrors( BDS_DSM_SET_FAILED_SINCE_CLEAR_MASK_DU16, ADR( DFES_numEntryAvl ) );
//appl_errList_s := bds_dsmDTC_getErrList(bds_dsmCmn_setFailedClrMsk_DU16, TRUE); 
//DFES_numEntryAvl := appl_errList_s.nrErr_u8;
bds_dsm_getErrors(BDS_DSM_SET_FAILED_SINCE_CLEAR_MASK_DU16, TRUE, 32, ADR(DFES_numEntryAvl), ADR(dfc_as));

(* check the DFES for error entries *)
IF (DFES_numEntryAvl > 0) THEN
    FOR cntrDfes_u8 := 0 TO (UINT_TO_USINT(DFES_numEntryAvl) - 1) DO
        ErrMemMgr_s.dtc_error_au32[cntrDfes_u8] := 0;
        ErrMemMgr_s.stDfes_au8[cntrDfes_u8]     := 0;
        ErrMemMgr_s.dfc_s.id                    := 0;
        idxActEntry_u8                          := ErrMemMgr_stNoEntryAvl_DU8;
        idxFirstEmptyEntry_u8                   := ErrMemMgr_stNoEntryAvl_DU8;
        (* get error status of DFES entries *)
        //ErrMemMgr_s.stDfes_au8[cntrDfes_u8] := (SHR(iDFC_st[iDFES_numDFC[cntrDfes_u8]], 3)) AND ErrMemMgr_BitMaskErrSts_DU8;
        dsmDTC_getStatus_s                  := bds_dsmDTC_getStatus(dfc_as[cntrDfes_u8].id);
        ErrMemMgr_s.stDfes_au8[cntrDfes_u8] := TO_USINT(dsmDTC_getStatus_s.errState_e);
        //bds_dsm_getDFC_Status(dfc_active_as[cntrDfes_u8],ADR(status_u16)); 
        //ErrMemMgr_s.stDfes_au8[cntrDfes_u8]:= UINT_TO_USINT(status_u16);
        IF (ErrMemMgr_s.stDfes_au8[cntrDfes_u8] <> 0) THEN (* DFES entry with error status found *)
            ErrMemMgr_s.nrDfesEntr_u8 := ErrMemMgr_s.nrDfesEntr_u8 + 1;
            ErrMemMgr_s.dfc_s.id      := dfc_as[cntrDfes_u8].id;
            ErrMemMgr_s.dfc_s.debmode := dfc_as[cntrDfes_u8].debmode;
            (* returns the DTC of a specified DFC *)
            ErrMemMgr_s.status_au16[cntrDfes_u8] := bds_dsm_getDTC_DFC(ErrMemMgr_s.dfc_s, ADR(ErrMemMgr_s.dtc_error_au32[cntrDfes_u8]));
            (* compare DTC with application buffer *)
            FOR cntrApplBuf_u8 := 0 TO ErrMemMgr_nrDfesEntries_DU8 - 1 DO
                (* check in application buffer if DTC is already listed *)
                IF (ErrMemMgr_s.ErrMemMgr_savePrm_s.ErrMemMgr_prevActvDfes_as[cntrApplBuf_u8].idxPrevActvDfes_u32 =
                   ErrMemMgr_s.dtc_error_au32[cntrDfes_u8]) AND
                   (idxActEntry_u8 = ErrMemMgr_stNoEntryAvl_DU8) THEN
                    idxActEntry_u8 := cntrApplBuf_u8; (* entry already available in application buffer *)
                ELSIF (ErrMemMgr_s.ErrMemMgr_savePrm_s.ErrMemMgr_prevActvDfes_as[cntrApplBuf_u8].idxPrevActvDfes_u32 = 0) AND
                      (idxFirstEmptyEntry_u8 = ErrMemMgr_stNoEntryAvl_DU8) THEN
                    idxFirstEmptyEntry_u8 := cntrApplBuf_u8; (* first empty entry in application buffer *)
                ELSE
                    ; (* entry not interesting *)
                END_IF;
            END_FOR;

            (* logic applied to get the previously active or deactive DTCs *)
            IF (((ErrMemMgr_s.stDfes_au8[cntrDfes_u8]) = bds_dsmCmn_stErrDeactv_e) OR (* Saved Errors *)
                ((ErrMemMgr_s.stDfes_au8[cntrDfes_u8]) = bds_dsmCmn_stErrPrevActv_e
                    ) OR (* Previously active errors (errors which healed during ECU-Reset) *)
                ((ErrMemMgr_s.stDfes_au8[cntrDfes_u8]) <> bds_dsmCmn_stErrActv_e
                    ) AND (* No active error (can be saved and active (Bit-Mask 0x07) *)
                (idxActEntry_u8 = ErrMemMgr_stNoEntryAvl_DU8) AND
                (idxFirstEmptyEntry_u8 <> ErrMemMgr_stNoEntryAvl_DU8)) THEN (*  no actual entry available and empty entry in buffer available *)
                (* collecting the previously active or deactive DTCs into application buffer *)
                ErrMemMgr_s.ErrMemMgr_savePrm_s.ErrMemMgr_prevActvDfes_as[idxFirstEmptyEntry_u8].idxPrevActvDfes_u32 :=
                    ErrMemMgr_s.dtc_error_au32[cntrDfes_u8];

                ErrMemMgr_s.ErrMemMgr_savePrm_s.ErrMemMgr_prevActvDfes_as[idxFirstEmptyEntry_u8].tiStamp_min_u32 := bds_sys_getAge();
                (* check DTCs if it is active again *)
            ELSIF ((ErrMemMgr_s.stDfes_au8[cntrDfes_u8]) = bds_dsmCmn_stErrActv_e) AND (* Active error *)
                  (idxActEntry_u8 <> ErrMemMgr_stNoEntryAvl_DU8) THEN                  (* actual entry available in buffer *)
                (*remove the active DTCs from the application buffer so as to hold only previously active or deactive DTCs*)
                ErrMemMgr_s.ErrMemMgr_savePrm_s.ErrMemMgr_prevActvDfes_as[idxActEntry_u8].idxPrevActvDfes_u32 := 0;
                ErrMemMgr_s.ErrMemMgr_savePrm_s.ErrMemMgr_prevActvDfes_as[idxActEntry_u8].tiStamp_min_u32     := 0;
            ELSE
                ; (* no error in DFES entry *)
            END_IF;
        END_IF;
    END_FOR;
END_IF
END_ACTION

END_PROGRAM

// BODAS_RC18_12_40/Application/00 Init/INIT_PRG
(*********************************************************************************************************************
 *     __   __   ___  ___           __   __        __   __  ___
 *   /_ / /  / /__  /    /__/     /_ / /_   |_ / /_ / /  /  /  /__/
 *  /__/ /__/ __ / /__  /  /     /  | /__  /  | /  | /__/  /  /  /
 *
 * Project: Hello World for ml290.rts
 *
 * Program: PLC_PRG
 *
 * Description:
 * PLC_PRG for initialization
 *
 * (c) Copyright by BOSCH REXROTH AG, all rights reserved
 *
 *********************************************************************************************************************)
PROGRAM INIT_PRG

VAR
	st_InitDone_b      : BOOL;
	ResetInfo_struc    : bds_ResetInfo_ts;
 	ResetInfoData_au32 : ARRAY[0..1] OF UDINT;
	
	ApplSwName_str     : STRING(50) := 'Hello World ml290.rts';

	UDSUUID_no_au8     : ARRAY[1..18] OF USINT;
	
	status_u16 : UINT;
END_VAR

IF( NOT( st_InitDone_b ) ) THEN 
	(******************************************************************************)
	(******************** Initialization: CAN communication  **********************)
	(******************************************************************************)
	INIT_initCAN();
	
	
	(******************************************************************************)
	(******************** Configuration: Input  ***********************************)
	(******************************************************************************)
	INIT_cfgInputs();
	
	
	(******************************************************************************)
	(******************** Configuration: Outputs **********************************)
	(******************************************************************************)
	INIT_cfgOutputs();
	
	
	(******************************************************************************)
	(******************** Initalization: UDS **************************************)
	(******************************************************************************)
	INIT_initUDS();
	
	
	(******************************************************************************)
	(******************** Initalization: NVM **************************************)
	(******************************************************************************)
	INIT_initNVM();
	
	
	(******************************************************************************)
	(******************** Initalization: General System****************************)
	(******************************************************************************)
	INIT_initSys();
	
	(******************** Initalization: Errors ***********************************)
	PRG_DebugManager.ACT_InitDebugManager();
	
	(* Set Init Done *)
	st_InitDone_b := TRUE;
	
END_IF

ACTION INIT_cfgInputs:
(******************************************************************************)
(******************** Initialization: Input  **********************************)
(******************************************************************************)
PRG_Inputs.ACT_InitInputs();
END_ACTION

ACTION INIT_cfgOutputs:
(******************************************************************************)
(******************** Initialization: Output  *********************************)
(******************************************************************************)

PRG_Outputs.ACT_InitOutputs();

(******************************************************************************)
(******************** Initialization: Safeout  ********************************)
(******************************************************************************)

PRG_SafeOuts.ACT_InitSafeOutputs();
END_ACTION

ACTION INIT_initCAN:
(*******************************************************************)
(******************** Initialization: CAN IN  **********************)
(*******************************************************************)
PRG_CANIn.ACT_InitCANIn();
(*******************************************************************)
(******************** Initialization: CAN OUT  *********************)
(*******************************************************************)
PRG_CANOut.ACT_InitCANOut();
(*******************************************************************)
(******************** Initialization: ISOBUS J1939  ****************)
(*******************************************************************)
PRG_ISOBUSJ1939.ACT_InitISOBUSJ1939();
END_ACTION

ACTION INIT_initNVM:
(******************************************************************************)
(******************** Initialization: NVM  ************************************)
(******************************************************************************)
bds_mem_readBlock(UINT_TO_USINT(bds_mem_nvmBlock01_512_R_D), ADR(GlobalVariables.PrmAsw_gstruc), 0, SIZEOF(GlobalVariables.PrmAsw_gstruc));
PRG_NVMConfig.ACT_InitNVMConfig();
END_ACTION

ACTION INIT_initSys:
(******************************************************************************)
(******************** Initialization: General System***************************)
(******************************************************************************)
(* --> debug: get reset info AND send it via CAN *)
bds_sys_getResetInfo(ADR(ResetInfo_struc)); (* reads the reset information of ECU *)
bds_can_sendData(bds_can_Chnl_te.BDS_CAN_2_D, 16#10001, BDS_CAN_EXD_DU8, 2, ADR(ResetInfo_struc.rbr_Grp_u16));
bds_can_sendData(bds_can_Chnl_te.BDS_CAN_2_D, 16#10002, BDS_CAN_EXD_DU8, 2, ADR(ResetInfo_struc.rbr_Type_u16));
ResetInfoData_au32[0] := ResetInfo_struc.rbr_UserDefined_u32;
bds_can_sendData(bds_can_Chnl_te.BDS_CAN_2_D, 16#10003, BDS_CAN_EXD_DU8, 4, ADR(ResetInfoData_au32));
(* debug <-- *)
(* ASW name AND HW-ID *)
bds_sys_applSwName(ADR(ApplSwName_str)); (* RC27-18/40 w/o Ethernet for others see the BSW manual *)
(* UUID (Byte 1..16) 392a682f-06fb-41eb-8b25-9b7ee48892f3 + major version (Byte 17) and minor version (Byte 18) *)
(* Defined in BODAS-service Editor *)
UDSUUID_no_au8[1]  := 16#39;
UDSUUID_no_au8[2]  := 16#2A;
UDSUUID_no_au8[3]  := 16#68;
UDSUUID_no_au8[4]  := 16#2F;
UDSUUID_no_au8[5]  := 16#06;
UDSUUID_no_au8[6]  := 16#FB;
UDSUUID_no_au8[7]  := 16#41;
UDSUUID_no_au8[8]  := 16#EB;
UDSUUID_no_au8[9]  := 16#8B;
UDSUUID_no_au8[10] := 16#25;
UDSUUID_no_au8[11] := 16#9B;
UDSUUID_no_au8[12] := 16#7E;
UDSUUID_no_au8[13] := 16#E4;
UDSUUID_no_au8[14] := 16#88;
UDSUUID_no_au8[15] := 16#92;
UDSUUID_no_au8[16] := 16#F3;
(* version *)
UDSUUID_no_au8[17] := 16#01; (* major version *)
UDSUUID_no_au8[18] := 16#23; (* minor version *)
(* Set UDS UUID for the BODAS-service App *)
bds_uds_setUUID(ADR(UDSUUID_no_au8[1]), 16);
(* Postrun and CAN Wakeup *)
bds_sys_requestPostRunProlong(); (* request for prolong in postrun *)
(* Enable writing and forcing *)
bds_codesys_setForcingWritingMode(16#FFFF);
END_ACTION

ACTION INIT_initUDS:
(******************************************************************************)
(******************** Initialization: UDS  ************************************)
(******************************************************************************)
PRG_UDS.ACT_InitUDS();
END_ACTION

END_PROGRAM

// BODAS_RC18_12_40/Application/01 MainTask/11 Parameters/PRG_DebugManager
(*********************************************************************************************************************
 *     __   __   ___  ___           __   __        __   __  ___
 *   /_ / /  / /__  /    /__/     /_ / /_   |_ / /_ / /  /  /  /__/
 *  /__/ /__/ __ / /__  /  /     /  | /__  /  | /  | /__/  /  /  /
 *
 * Project: Hello World for ml290.rts
 *
 * Program: PRG_DebugManager
 *
 * Author:  
 *
 * Description:
 * Interface for Debug Manager
 *
 * (c) Copyright by BOSCH REXROTH AG, all rights reserved
 *
 *********************************************************************************************************************)
PROGRAM PRG_DebugManager
VAR
	DbgMgr_struc : struc_DbgMgr; 
END_VAR

IF( DbgMgr_struc.prm_struc.flgXcpOn_b) THEN
  (* enable XCP *)
  bds_xcp_setMode(BDS_ENABLE_XCP_DU16);

ELSE
  (* disable XCP *)
  bds_xcp_setMode(BDS_DISABLE_XCP_DU16);

END_IF

(* Recognise a rising edge *)
DbgMgr_struc.outp_struc.flgStoreDataToNvmReq_l := FUNC_DbgMgrRisingEdgeDetn(i_curr_b:= DbgMgr_struc.prm_struc.flgStoreDataToNvm_b, i_prev_pb:= ADR(DbgMgr_struc.prv_struc.flgStoreDataToNvmPrev_l) );

(* Save parameters in Nvm if requested via XCP *)
IF( DbgMgr_struc.outp_struc.flgStoreDataToNvmReq_l ) THEN
	(* PrmMgr_SaveNvmAll(); todo *)
	
	(* Get lock so parameters are not modified during copy to Nvm RAM (e.g. UDS/XCP) *)
	BDS_SYS_GET_LOCK_COMMON();
	
	(* copy ram mirror of block 1 into NVM todo report stsSaveFct_u16 *)
	bds_mem_writeBlock(UINT_TO_USINT(bds_mem_nvmBlock02_512_R_D), ADR(DbgMgr_struc), 0, SIZEOF(DbgMgr_struc));
	
	(* Release lock *)
	BDS_SYS_RELEASE_LOCK_COMMON();

END_IF

ACTION ACT_InitDebugManager:
  DbgMgr_struc.prv_struc.flgStoreDataToNvmPrev_l := 0;
  DbgMgr_struc.outp_struc.flgStoreDataToNvmReq_l := 0;

  IF(DbgMgr_struc.prm_struc.flgXcpOn_b) THEN  
      (* enable XCP *)
      bds_xcp_setMode(BDS_ENABLE_XCP_DU16);
    
  END_IF
END_ACTION

END_PROGRAM

// BODAS_RC18_12_40/Application/01 MainTask/11 Parameters/Functions/FUNC_DbgMgrRisingEdgeDetn
FUNCTION FUNC_DbgMgrRisingEdgeDetn : BOOL
VAR_INPUT
	i_curr_b : BOOL;
	i_prev_pb : POINTER TO BOOL;
END_VAR
VAR
	retval_b : BOOL;
END_VAR

(* Check if current value is true but previous value was false *)
IF( i_curr_b AND NOT(i_prev_pb^) ) THEN
	retval_b := TRUE;

ELSE
	retval_b := FALSE;

END_IF	

(* Make backup copy of current value *)
i_prev_pb^ := i_curr_b;

FUNC_DbgMgrRisingEdgeDetn := retval_b;

END_FUNCTION

// BODAS_RC18_12_40/Application/01 MainTask/02 Outputs/PRG_SafeOuts
(*********************************************************************************************************************
*    __   __   ___  ___           __   __        __   __  ___
*   /_ / /  / /__  /    /__/     /_ / /_   |_ / /_ / /  /  /  /__/
*  /__/ /__/ __ / /__  /  /     /  | /__  /  | /  | /__/  /  /  /
*
* Project: Hello World for ml290.rts
*
* Program: PRG_Outputs
*
* Author:  
*
* Description:
* Interface for the hardware outputs to the application
*
* (c) Copyright by BOSCH REXROTH AG, all rights reserved
*
*********************************************************************************************************************)
PROGRAM PRG_SafeOuts
VAR
    PHMDL_CHNL1 : UINT := UDINT_TO_UINT(PHMDL OR CHNL1);
END_VAR

ACTION ACT_InitSafeOutputs:
(*configure SAFOUT with PHMDL mode (HS1 - K09, HS2 - K73 AND LS - K14)*)
bds_out_po_cfg(bds_out_po_signal_te.K09, STD_ON); (* Configure K09 for POC *)
bds_out_po_cfg(bds_out_po_signal_te.K73, STD_ON); (* Configure K73 for POC *)
bds_safout_cfg(UDINT_TO_UINT(PHMDL_CHNL1),
               bds_out_po_signal_te.K14,
               bds_out_po_signal_te.K09,
               bds_out_po_signal_te.K73,
               0,
               0);
END_ACTION

END_PROGRAM

// BODAS_RC18_12_40/Application/01 MainTask/03 Communication/01 ISOBUSJ1939/PRG_ISOBUSJ1939
(*********************************************************************************************************************
 *     __   __   ___  ___           __   __        __   __  ___
 *   /_ / /  / /__  /    /__/     /_ / /_   |_ / /_ / /  /  /  /__/
 *  /__/ /__/ __ / /__  /  /     /  | /__  /  | /  | /__/  /  /  /
 *
 * Project: Hello World for ml290.rts
 *
 * Program: PRG_ISOBUSJ1939
 *
 * Author:  
 *
 * Description:
 * Interface for ISOBUS
 *
 * (c) Copyright by BOSCH REXROTH AG, all rights reserved
 *
 *********************************************************************************************************************)
PROGRAM PRG_ISOBUSJ1939
VAR
    dataJ1939Inst_as       : ARRAY[1..enu_IsobusJ1939_IsobusInst.IsobusJ1939_IsobusInstMax_E] OF bds_isobus_appInst_ts;
    dataTxBufDataBoxes1_as : ARRAY[1..enu_IsobusJ1939_TxInst1Box.IsobusJ1939_TxInst1BoxMax_E] OF bds_isobus_txMsg_ts;
    dataRxBufDataBoxes1_as : ARRAY[1..enu_IsobusJ1939_RxInst1Box.IsobusJ1939_RxInst1BoxMax_E] OF bds_isobus_rxMsg_ts;
    dataTxBufDataBoxes2_as : ARRAY[1..enu_IsobusJ1939_TxInst2Box.IsobusJ1939_TxInst2BoxMax_E] OF bds_isobus_txMsg_ts;
    dataRxBufDataBoxes2_as : ARRAY[1..enu_IsobusJ1939_RxInst2Box.IsobusJ1939_RxInst2BoxMax_E] OF bds_isobus_rxMsg_ts;
    dataTxBufDataBoxes3_as : ARRAY[1..enu_IsobusJ1939_TxInst3Box.IsobusJ1939_TxInst3BoxMax_E] OF bds_isobus_txMsg_ts;
    dataRxBufDataBoxes3_as : ARRAY[1..enu_IsobusJ1939_RxInst3Box.IsobusJ1939_RxInst3BoxMax_E] OF bds_isobus_rxMsg_ts;
    dataJ1939Dm1Failrs_as  : ARRAY[1..86] OF bds_isobus_dtcList_ts; (* failure list struct-array *)
END_VAR

;

END_PROGRAM

// BODAS_RC18_12_40/Application/01 MainTask/10 Service/PRG_UDS
(*********************************************************************************************************************
 *     __   __   ___  ___           __   __        __   __  ___
 *   /_ / /  / /__  /    /__/     /_ / /_   |_ / /_ / /  /  /  /__/
 *  /__/ /__/ __ / /__  /  /     /  | /__  /  | /  | /__/  /  /  /
 *
 * Project: Hello World for ml321.rts
 *
 * Program: PLC_UDS
 *
 * Description:
 * PLC_PRG for initialisation
 *
 * (c) Copyright by BOSCH REXROTH AG, all rights reserved
 *
 *********************************************************************************************************************)
PROGRAM PRG_UDS
VAR
END_VAR

;

ACTION ACT_InitUDS:
(******************************************************************************)
(******************** Register UDS Callback  **********************************)
(******************************************************************************)
bds_uds_registerDidReadCallback(ADR(UDS_ReadCallback));
bds_uds_registerDidWriteCallback(ADR(UDS_WriteCallback));
bds_uds_registerRoutineF000Callback(ADR(UDS_RoutineCallback));
bds_uds_registerRoutineF001Callback(ADR(UDS_DefaultCallback));
END_ACTION

END_PROGRAM

// BODAS_RC18_12_40/Application/01 MainTask/10 Service/Programs/UDS_ReadCallback
FUNCTION UDS_ReadCallback
VAR_INPUT
    //a variable to which the content has to be written
    UDSReadData_pau8 : POINTER TO USINT;
END_VAR
VAR
    // variables for internal operations
    //data_au8 : ARRAY[0..8] OF BYTE;
    i                     : BYTE;
    DidValue_u16          : UINT;
    set_u8                : USINT;
    ret_secLevel          : UINT;
    Level_pu16            : POINTER TO UINT;
    ret_response          : BOOL;
    temp_sec_level        : BOOL;
    uPmpSnsr_mV_u16       : UINT;
    fctPmp_s16            : INT;
    stBrkSwt_u8           : USINT;
    iPmpFwdAct_mA_u16     : UINT;
    funcRet_u8            : USINT;
    UDSReadData_pau8_poby : POINTER TO ARRAY[0..7] OF BYTE;
    UDSReadData_pau8_by   : ARRAY[0..7] OF BYTE;
    DID_0103_s32          : DINT;
    DiagChkLvlRet_u8      : USINT;
END_VAR

(* Get the DID requested by tester present *)
bds_uds_GetActiveDid(ADR(DidValue_u16));

//bds_can_sendData(bds_can_Chnl_te.BDS_CAN_1_D, 5, BDS_CAN_EXD_DU8, 2, ADR(DidValue_u16));
//CASE DidValue_u16 OF
// 16#C003, 16#D001, 16#D002:
(* here check th security level *)
//bds_sec_getLevel(BDS_SEC_ASW_INST_NAME_2_E, ADR(Level_pu16));
//DiagChkLvlRet_u8 := UDS_Diag_ChkLvl(16#00000004, Level_pu16^);
//ELSE
(* all levels allowed *)
//bds_sec_getLevel(BDS_SEC_ASW_INST_NAME_1_E, ADR(Level_pu16));
//DiagChkLvlRet_u8 := UDS_Diag_ChkLvl(16#FFFFFFFF, Level_pu16^);
//DiagChkLvlRet_u8 := 0;
//END_CASE
IF (TRUE) THEN
    //IF( NOT( USINT_TO_BOOL( DiagChkLvlRet_u8 ) ) ) THEN 
    CASE DidValue_u16 OF
    (* Handle the read operation at DIDs *)
    (* Parameters *)
    16#C001: bds_uds_setCallbackStatus(0); (* E_OK *)
        UDSReadData_pau8[1] := INT_TO_BYTE(SHR(GlobalVariables.PrmAsw_gstruc.fctPmp_s16, 8));
        UDSReadData_pau8[0] := INT_TO_BYTE(GlobalVariables.PrmAsw_gstruc.fctPmp_s16);
    16#C002: bds_uds_setCallbackStatus(0); (* E_OK *)
        UDSReadData_pau8[1] := TO_BYTE(SHR(GlobalVariables.PrmAsw_gstruc.listCtrlVlv_enu, 8));
        UDSReadData_pau8[0] := TO_BYTE(GlobalVariables.PrmAsw_gstruc.listCtrlVlv_enu);
    16#C003: bds_uds_setCallbackStatus(0); (* E_OK *)
        UDSReadData_pau8[1] := INT_TO_BYTE(SHR(GlobalVariables.PrmAsw_gstruc.nrCogs_s16, 8));
        UDSReadData_pau8[0] := INT_TO_BYTE(GlobalVariables.PrmAsw_gstruc.nrCogs_s16);
    16#01C7: bds_uds_setCallbackStatus(0); (* E_OK *)
        UDSReadData_pau8[1] := UINT_TO_BYTE(SHR(GlobalVariables.PrmAsw_gstruc.iSpSafout1_u16, 8));
        UDSReadData_pau8[0] := UINT_TO_BYTE(GlobalVariables.PrmAsw_gstruc.iSpSafout1_u16);
    16#01C8: bds_uds_setCallbackStatus(0); (* E_OK *)
        UDSReadData_pau8[1] := UINT_TO_BYTE(SHR(GlobalVariables.PrmAsw_gstruc.iSpSafout2_u16, 8));
        UDSReadData_pau8[0] := UINT_TO_BYTE(GlobalVariables.PrmAsw_gstruc.iSpSafout2_u16);
    16#D001: bds_uds_setCallbackStatus(0); (* E_OK *)
        UDSReadData_pau8[0] := BOOL_TO_BYTE(GlobalVariables.PrmAsw_gstruc.PrmDbg_struc.flgXcpOn_b);
    16#D002: bds_uds_setCallbackStatus(0); (* E_OK *)
        UDSReadData_pau8[0] := BOOL_TO_BYTE(GlobalVariables.PrmAsw_gstruc.PrmDbg_struc.flgStoreDataToNvm_b);
    16#C010: bds_uds_setCallbackStatus(0); (* E_OK *)
        UDSReadData_pau8[1] := UINT_TO_BYTE(SHR(GlobalVariables.PrmAsw_gstruc.eff_perc_au16[0], 8));
        UDSReadData_pau8[0] := UINT_TO_BYTE(GlobalVariables.PrmAsw_gstruc.eff_perc_au16[0]);
        UDSReadData_pau8[3] := UINT_TO_BYTE(SHR(GlobalVariables.PrmAsw_gstruc.eff_perc_au16[1], 8));
        UDSReadData_pau8[2] := UINT_TO_BYTE(GlobalVariables.PrmAsw_gstruc.eff_perc_au16[1]);
        UDSReadData_pau8[5] := UINT_TO_BYTE(SHR(GlobalVariables.PrmAsw_gstruc.eff_perc_au16[2], 8));
        UDSReadData_pau8[4] := UINT_TO_BYTE(GlobalVariables.PrmAsw_gstruc.eff_perc_au16[2]);
    16#C020: bds_uds_setCallbackStatus(0); (* E_OK *)
        UDSReadData_pau8[1] := UINT_TO_BYTE(SHR(GlobalVariables.PrmAsw_gstruc.nEngSpd_rpm_au16[0], 8));
        UDSReadData_pau8[0] := UINT_TO_BYTE(GlobalVariables.PrmAsw_gstruc.nEngSpd_rpm_au16[0]);
        UDSReadData_pau8[3] := UINT_TO_BYTE(SHR(GlobalVariables.PrmAsw_gstruc.nEngSpd_rpm_au16[1], 8));
        UDSReadData_pau8[2] := UINT_TO_BYTE(GlobalVariables.PrmAsw_gstruc.nEngSpd_rpm_au16[1]);
        UDSReadData_pau8[5] := UINT_TO_BYTE(SHR(GlobalVariables.PrmAsw_gstruc.nEngSpd_rpm_au16[2], 8));
        UDSReadData_pau8[4] := UINT_TO_BYTE(GlobalVariables.PrmAsw_gstruc.nEngSpd_rpm_au16[2]);
    (* Process Values *)
    16#A001: bds_uds_setCallbackStatus(0); (* E_OK *)
        UDSReadData_pau8[1] := UINT_TO_BYTE(SHR(PRG_Inputs.uPmpSnsr_mV_u16, 8));
        UDSReadData_pau8[0] := UINT_TO_BYTE(PRG_Inputs.uPmpSnsr_mV_u16);
    16#A002: bds_uds_setCallbackStatus(0); (* E_OK *)
        UDSReadData_pau8[0] := INT_TO_BYTE(PRG_Outputs.st_BrkSwt_u8);
    16#A003: bds_uds_setCallbackStatus(0); (* E_OK *)
        UDSReadData_pau8[1] := UDINT_TO_BYTE(SHR(PRG_Inputs.frqVehSnsr_Hz_u32, 8));
        UDSReadData_pau8[0] := UDINT_TO_BYTE(PRG_Inputs.frqVehSnsr_Hz_u32);
    16#B001: bds_uds_setCallbackStatus(0); (* E_OK *)
        UDSReadData_pau8[1] := UINT_TO_BYTE(SHR(PRG_Outputs.no_CurrentK07_mA_u16, 8));
        UDSReadData_pau8[0] := UINT_TO_BYTE(PRG_Outputs.no_CurrentK07_mA_u16);
    16#B002: bds_uds_setCallbackStatus(0); (* E_OK *)
        UDSReadData_pau8[0] := PRG_Outputs.st_CtrlValve_u8;
    16#B003: bds_uds_setCallbackStatus(0); (* E_OK *)
        UDSReadData_pau8[1] := UINT_TO_BYTE(SHR(PRG_Inputs.vWhlSpd_kph_u16, 8));
        UDSReadData_pau8[0] := UINT_TO_BYTE(PRG_Inputs.vWhlSpd_kph_u16);
        ELSE
            bds_uds_setCallbackStatus(1); (* E_OK *)
    END_CASE
ELSE
    bds_uds_setCallbackStatus(1); (* E_NOK *)
END_IF

END_FUNCTION

// BODAS_RC18_12_40/Application/01 MainTask/10 Service/Programs/UDS_Diag_ChkLvl
(*********************************************************************************************************************
 *     __   __   ___  ___           __   __        __   __  ___
 *   /_ / /  / /__  /    /__/     /_ / /_   |_ / /_ / /  /  /  /__/
 *  /__/ /__/ __ / /__  /  /     /  | /__  /  | /  | /__/  /  /  /
 *
 * Project: Hello World for ml290.rts
 *
 * Function: UDS_Diag_ChkLvl
 *
 * Author:  
 *
 * Description:
 * Function for level check
 *
 * (c) Copyright by BOSCH REXROTH AG, all rights reserved
 *
 *********************************************************************************************************************)
FUNCTION UDS_Diag_ChkLvl : USINT
VAR_INPUT
    i_Mask_u32  : UDINT;
    i_Level_u16 : UINT;
END_VAR

(*UDS_Diag_ChkLvl := GVL_UDS.UDS_NEGATIVE_RESPONSE;*)
UDS_Diag_ChkLvl := 1;

(* First check security as defined in ISO 14229 - see bds_sec_accessLevel_te *)
IF (0 <> (UDINT_TO_WORD(i_Mask_u32) AND SHL(i_Level_u16, 16#1))) THEN
    (*UDS_Diag_ChkLvl := GVL_UDS.UDS_POSITIVE_RESPONSE;*)
    UDS_Diag_ChkLvl := 0;
ELSE
    ;
END_IF

END_FUNCTION

// BODAS_RC18_12_40/Application/01 MainTask/10 Service/Programs/UDS_WriteCallback
FUNCTION UDS_WriteCallback
VAR_INPUT
    UDSReadData_pau8 : POINTER TO USINT;
END_VAR
VAR
    DidValue_u16     : UINT;
    DiagChkLvlRet_u8 : USINT;
    Level_pu8        : POINTER TO USINT;
END_VAR

(* Get the DID requested by tester present *)
bds_uds_GetActiveDid(ADR(DidValue_u16));

(* here check the security level *)
CASE DidValue_u16 OF
16#C003, 16#D001, 16#D002:
    (* security level 2 *)
    //bds_sec_getLevel(BDS_SEC_ASW_INST_NAME_1_E, ADR(Level_pu8));
    //DiagChkLvlRet_u8 := UDS_Diag_ChkLvl(16#00000004, Level_pu8^);
    DiagChkLvlRet_u8 := 0;
    ELSE
        (*bds_sec_getLevel(BDS_SEC_ASW_INST_NAME_1_E, ADR(Level_pu8));
	DiagChkLvlRet_u8 := UDS_Diag_ChkLvl(16#FFFFFFFF, Level_pu8^);*)
        DiagChkLvlRet_u8 := 0;
END_CASE

IF (NOT (USINT_TO_BOOL(DiagChkLvlRet_u8))) THEN
    CASE DidValue_u16 OF
    (* Handle the write operation at DID 0xC001 *)
    16#C001: bds_uds_setCallbackStatus(0); (* E_OK *)
        GlobalVariables.PrmAsw_gstruc.fctPmp_s16 := WORD_TO_INT(USINT_TO_WORD(UDSReadData_pau8[0]) + SHL(USINT_TO_WORD(UDSReadData_pau8[1]), 8));
    (* Handle the write operation at DID 0xC002 *)
    16#C002: bds_uds_setCallbackStatus(0); (* E_OK *)
        GlobalVariables.PrmAsw_gstruc.listCtrlVlv_enu.0 := UDSReadData_pau8[0].0;
        GlobalVariables.PrmAsw_gstruc.listCtrlVlv_enu.1 := UDSReadData_pau8[0].1;
        GlobalVariables.PrmAsw_gstruc.listCtrlVlv_enu.2 := UDSReadData_pau8[0].2;
        GlobalVariables.PrmAsw_gstruc.listCtrlVlv_enu.3 := UDSReadData_pau8[0].3;
        GlobalVariables.PrmAsw_gstruc.listCtrlVlv_enu.4 := UDSReadData_pau8[0].4;
        GlobalVariables.PrmAsw_gstruc.listCtrlVlv_enu.5 := UDSReadData_pau8[0].5;
        GlobalVariables.PrmAsw_gstruc.listCtrlVlv_enu.6 := UDSReadData_pau8[0].6;
        GlobalVariables.PrmAsw_gstruc.listCtrlVlv_enu.7 := UDSReadData_pau8[0].7;
    (* Handle the write operation at DID 0xC003 *)
    16#C003: bds_uds_setCallbackStatus(0); (* E_OK *)
        GlobalVariables.PrmAsw_gstruc.nrCogs_s16 := WORD_TO_INT(USINT_TO_WORD(UDSReadData_pau8[0]) + SHL(USINT_TO_WORD(UDSReadData_pau8[1]), 8));
    (* Handle the write operation at DID 0x01C7 *)
    16#01C7: bds_uds_setCallbackStatus(0); (* E_OK *)
        GlobalVariables.PrmAsw_gstruc.iSpSafout1_u16 :=
            WORD_TO_UINT(USINT_TO_WORD(UDSReadData_pau8[0]) + SHL(USINT_TO_WORD(UDSReadData_pau8[1]), 8));
    (* Handle the write operation at DID 0x01C8 *)
    16#01C8: bds_uds_setCallbackStatus(0); (* E_OK *)
        GlobalVariables.PrmAsw_gstruc.iSpSafout2_u16 :=
            WORD_TO_UINT(USINT_TO_WORD(UDSReadData_pau8[0]) + SHL(USINT_TO_WORD(UDSReadData_pau8[1]), 8));
    (* Handle the write operation at DID 0xD001 *)
    16#D001: bds_uds_setCallbackStatus(0); (* E_OK *)
        GlobalVariables.PrmAsw_gstruc.PrmDbg_struc.flgXcpOn_b := USINT_TO_BOOL(UDSReadData_pau8[0]);
    (* Handle the write operation at DID 0xD002 *)
    16#D002: bds_uds_setCallbackStatus(0); (* E_OK *)
        GlobalVariables.PrmAsw_gstruc.PrmDbg_struc.flgStoreDataToNvm_b := USINT_TO_BOOL(UDSReadData_pau8[0]);
    (* Handle the write operation at DID 0xC010 *)
    16#C010: bds_uds_setCallbackStatus(0); (* E_OK *)
        //GlobalVariables.PrmAsw_gstruc.eff_perc_au16[0] := WORD_TO_UINT(USINT_TO_WORD(UDSReadData_pau8[0]) + SHL(USINT_TO_WORD(UDSReadData_pau8[1]), 8));
        //GlobalVariables.PrmAsw_gstruc.eff_perc_au16[1] := WORD_TO_UINT(USINT_TO_WORD(UDSReadData_pau8[2]) + SHL(USINT_TO_WORD(UDSReadData_pau8[3]), 8));
        //GlobalVariables.PrmAsw_gstruc.eff_perc_au16[2] := WORD_TO_UINT(USINT_TO_WORD(UDSReadData_pau8[4]) + SHL(USINT_TO_WORD(UDSReadData_pau8[5]), 8));
    (* Handle the write operation at DID 0xC020 *)
    16#C020:
            //GlobalVariables.PrmAsw_gstruc.nEngSpd_rpm_au16[0] := WORD_TO_UINT(USINT_TO_WORD(UDSReadData_pau8[0]) + SHL(USINT_TO_WORD(UDSReadData_pau8[1]), 8));
            //GlobalVariables.PrmAsw_gstruc.nEngSpd_rpm_au16[1] := WORD_TO_UINT(USINT_TO_WORD(UDSReadData_pau8[2]) + SHL(USINT_TO_WORD(UDSReadData_pau8[3]), 8));
            //GlobalVariables.PrmAsw_gstruc.nEngSpd_rpm_au16[2] := WORD_TO_UINT(USINT_TO_WORD(UDSReadData_pau8[4]) + SHL(USINT_TO_WORD(UDSReadData_pau8[5]), 8));
        ELSE
            bds_uds_setCallbackStatus(1); (* E_NOK *)
    END_CASE
ELSE
    bds_uds_setCallbackStatus(1); (* E_NOK *)
END_IF

END_FUNCTION

// BODAS_RC18_12_40/Application/01 MainTask/10 Service/Programs/UDS_RoutineCallback
PROGRAM UDS_RoutineCallback
VAR
    NvmWriteRet_u16  : UINT;
    DiagChkLvlRet_u8 : USINT;
    Level_pu8        : POINTER TO USINT;
END_VAR

(* here check th security level *)
//bds_sec_getLevel(BDS_SEC_ASW_INST_NAME_1_E, ADR(Level_pu8));
//DiagChkLvlRet_u8 := UDS_Diag_ChkLvl(16#00000004, Level_pu8^);
DiagChkLvlRet_u8 := 0;

IF (NOT (USINT_TO_BOOL(DiagChkLvlRet_u8))) THEN
    NvmWriteRet_u16 :=
        bds_mem_writeBlock(UINT_TO_USINT(bds_mem_nvmBlock01_512_R_D), ADR(GlobalVariables.PrmAsw_gstruc), 0, SIZEOF(GlobalVariables.PrmAsw_gstruc));

    IF (0 = NvmWriteRet_u16) THEN
        bds_uds_setCallbackStatus(0); (* E_OK *)
    ELSE
        bds_uds_setCallbackStatus(10); (* E_NOK which decrements to 1. i.e executes for 10 cycles before E_NOK is set ( wait time ill date is written to NVM) *)
    END_IF
ELSE
    bds_uds_setCallbackStatus(10); (* E_NOK *)
END_IF

END_PROGRAM

// BODAS_RC18_12_40/Application/01 MainTask/10 Service/Programs/UDS_DefaultCallback
PROGRAM UDS_DefaultCallback
VAR
END_VAR

GlobalVariables.PrmAsw_gstruc.fctPmp_s16                       := GlobalVariables.PrmAsw_cgstruc.fctPmp_s16;
GlobalVariables.PrmAsw_gstruc.listCtrlVlv_enu                  := GlobalVariables.PrmAsw_cgstruc.listCtrlVlv_enu;
GlobalVariables.PrmAsw_gstruc.nrCogs_s16                       := GlobalVariables.PrmAsw_cgstruc.nrCogs_s16;
GlobalVariables.PrmAsw_gstruc.iSpSafout1_u16                   := GlobalVariables.PrmAsw_cgstruc.iSpSafout1_u16;
GlobalVariables.PrmAsw_gstruc.iSpSafout2_u16                   := GlobalVariables.PrmAsw_cgstruc.iSpSafout2_u16;
GlobalVariables.PrmAsw_gstruc.PrmDbg_struc.flgXcpOn_b          := GlobalVariables.PrmAsw_cgstruc.PrmDbg_struc.flgXcpOn_b;
GlobalVariables.PrmAsw_gstruc.PrmDbg_struc.flgStoreDataToNvm_b := GlobalVariables.PrmAsw_cgstruc.PrmDbg_struc.flgStoreDataToNvm_b;
GlobalVariables.PrmAsw_gstruc.eff_perc_au16[0]                 := GlobalVariables.PrmAsw_cgstruc.eff_perc_au16[0];
GlobalVariables.PrmAsw_gstruc.eff_perc_au16[1]                 := GlobalVariables.PrmAsw_cgstruc.eff_perc_au16[1];
GlobalVariables.PrmAsw_gstruc.eff_perc_au16[2]                 := GlobalVariables.PrmAsw_cgstruc.eff_perc_au16[2];
GlobalVariables.PrmAsw_gstruc.nEngSpd_rpm_au16[0]              := GlobalVariables.PrmAsw_cgstruc.nEngSpd_rpm_au16[0];
GlobalVariables.PrmAsw_gstruc.nEngSpd_rpm_au16[1]              := GlobalVariables.PrmAsw_cgstruc.nEngSpd_rpm_au16[1];
GlobalVariables.PrmAsw_gstruc.nEngSpd_rpm_au16[2]              := GlobalVariables.PrmAsw_cgstruc.nEngSpd_rpm_au16[2];

END_PROGRAM
